// TIA Portal V18 export
TYPE "AnalogChannel_v0"
// stored: IsFailsafeCompliant false
   STRUCT
      CHRlyIsOn : Array[0..11] of Bool;   // Off/On
      CHRlyIsOff : Array[0..11] of Bool;   // Off/On
      CHRlyOnCmd : Array[0..11] of Bool;   // Off/On
      CHInitialSignal : Array[0..11] of Real;   // 0-100.0%
      CHAdaptedSignal : Array[0..11] of Real;   // 0-100.0%
   END_STRUCT;
END_TYPE
